Fanuc KAREL source: IO0108.KL

PROGRAM IO0108
%STACKSIZE=65535
%PRIORITY=65535
%NOLOCKGROUP
ROUTINE RTEST FROM IO0108
ROUTINE RTEST
VAR
L1 : ARRAY[3] OF INTEGER
L2 : XYZWPR
L3 : JOINTPOS9
L4 : POSITION
U2C_37 : BOOLEAN
U2C_38 : REAL
U2C_39 : REAL
U2C_40 : INTEGER
U2C_41 : REAL
BEGIN
U2C_37=TRUE
L1[1]=2
U2C_40=1
U2C_41=1.0
-- UNRESOLVED_PC line 19 opcodes [21 9D 1A] marker_code=77
END RTEST
BEGIN
RTEST
END IO0108
